// TIA Portal V18 export
// export: Created 2025-12-01T17:53:10.286845Z, ExportSetting None, DisplayName Totally Integrated Automation Portal, DisplayVersion V18 Update 5, DisplayName TIA Portal Openness, DisplayVersion V18 Update 5, DisplayName TIA Portal Teamcenter Gateway, DisplayVersion V18, DisplayName TIA Portal Version Control Interface, DisplayVersion V18, DisplayName STEP 7 Professional, DisplayVersion V18 Update 5, DisplayName STEP 7 Safety, DisplayVersion V18, DisplayName WinCC Professional, DisplayVersion V18 Update 5
Screen "620SysDiagnosis"  1280x800, Number=620, Template=06Diagnosis
  ScreenLayer 
    Button "btnMenu7" at 768,725 size 128x75  StyleItem=BtnActive20, TextOff="系统诊断 / System Diagnosis / Sústava Diagnóza"
      on Press: ActivateScreen(Screen name := , Object number := 0); SetTag(Tag := Sys_VersionManagement_HMIPageID, Value := 620)
